Staubli VAL3: copy_folder.pgx

program copy_folder(string x_sPathCopy, string x_sPathPaste)
  local string l_sPathCopy
  local string l_sPathPaste
  local bool l_bCheck
  local num i
  local num j
  local string l_sEmpty
begin
  //
  // copy or not the x_sPathCopy to x_sPath
  //
  call use:timerDialog("Copying file: ##",0)
  call use:stringCopy(l_sEmpty,sPathSession)
  // all the folder are created
  if x_sPathCopy==""
    // copy from the template session
    l_sPathCopy="Disk://kernel/template/session/"
  else
    // copy form the x_sPathCopy session name
    l_sPathCopy="Disk://session/"+x_sPathCopy+"/"
  endIf
  // scan it
  l_bCheck=libList(l_sPathCopy,sPathSession)
  // copy form the x_sPathCopy session name
  l_sPathPaste="Disk://session/"+x_sPathPaste+"/"
  // start the copy
  for i=0 to size(sPathSession)-1
    // for all the directory found only one level...
    l_sEmpty=""
    call use:stringCopy(l_sEmpty,sDeeperSession)
    // scan the folder
    l_bCheck=libList(l_sPathCopy+sPathSession[i],sDeeperSession)
    for j=0 to size(sDeeperSession)-1
      // copy all the file
      call use:typeLen(1,6,l_sPathCopy+sPathSession[i]+"/"+sDeeperSession[j],38)
      call use:typeLen(1,7,l_sPathPaste+sPathSession[i]+"/"+sDeeperSession[j],38)
      l_bCheck=$copy(l_sPathCopy+sPathSession[i]+"/"+sDeeperSession[j],l_sPathPaste+sPathSession[i]+"/"+sDeeperSession[j])
      delay(0)
    endFor
    delay(0)
  endFor
end
